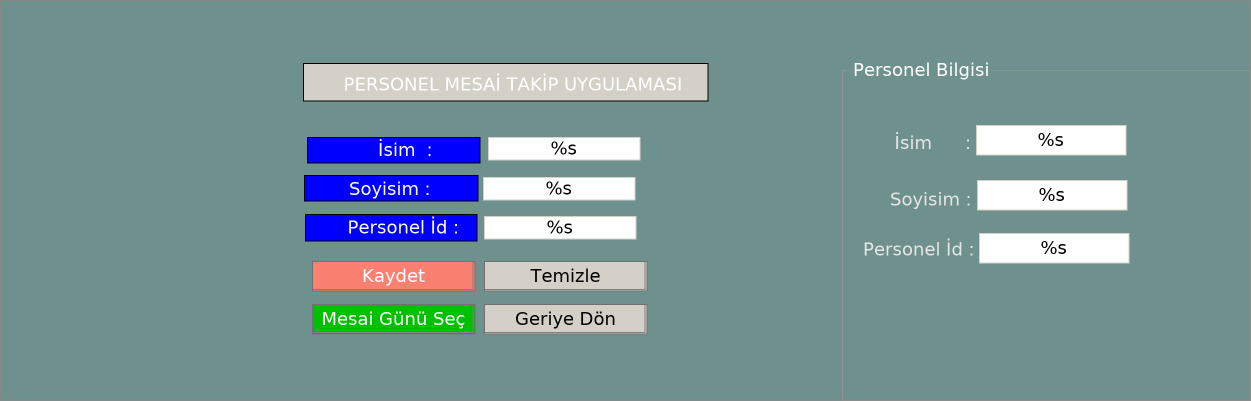
VISUALIZATION Kayit_Sayfa  // 1251x401
    Rectangle (305,214 172x27)
    Rectangle (303,63 405x38)
    Rectangle (307,137 173x26)
    Rectangle (304,175 174x26)
    Textfield (488,137 152x23), "%s", text variable: GVL_personel_kayit.perisim
        OnMouseClick: write the text variable via Edit
    Label (294,176 192x26), "Soyisim :"
    Label (323,132 165x36), "İsim :"
    Textfield (483,177 152x23), "%s", text variable: GVL_personel_kayit.perSoyisim
        OnMouseClick: write the text variable via Edit
    Label (315,71 396x27), "PERSONEL MESAİ TAKİP UYGULAMASI"
    Label (338,213 131x29), "Personel İd :"
    Textfield (484,216 152x23), "%s", text variable: GVL_personel_kayit.perid
        OnMouseClick: write the text variable via Edit
    Button (312,261 163x30), "Kaydet"
        tap GVL_personel_kayit.kaydet
        OnMouseClick: OpenDialog Dialog=VisuDialogs.MessageBox, Parameters={eType: GVL_personel_kayit.msgtype, sMessageTxt: GVL_personel_kayit.messagetext, sTitle: GVL_personel_kayit.messagetitle}, OpenModal=True, OpenCentered=True
    GroupBox (842,62 409x339), "Personel Bilgisi"
        Label (16,66 150x30), "İsim :"
        Label (14,123 150x29), "Soyisim :"
        Label (2,172 150x31), "Personel İd :"
        Textfield (135,118 150x30), "%s", text variable: GVL_personel_kayit.perSoyisim
            OnMouseClick: write the text variable via Edit
        Textfield (137,171 150x30), "%s", text variable: GVL_personel_kayit.perid
            OnMouseClick: write the text variable via Edit
        Textfield (134,63 150x30), "%s", text variable: GVL_personel_kayit.perisim
            OnMouseClick: write the text variable via Edit
    Button (312,304 163x30), "Mesai Günü Seç", invisible if: NOT GVL_personel_kayit.invisibleKayit
        tap GVL_personel_kayit.perMesaiGun
        OnMouseClick: change screen: mesaigunleri_sayfa
    Button (484,261 163x30), "Temizle"
        tap GVL_personel_kayit.temizle
    Button (484,304 163x30), "Geriye Dön"
        OnMouseClick: change screen: Ana_Sayfa
END_VISUALIZATION

(* stored: Version 1.1.0.1, ProductVersion 3.1.4024.12
   Visu Kayit_Sayfa: Id {fe354db6-dd9b-4736-b1f6-b1825fe609fa} *)
